FUNCTION_BLOCK Test_ListCountIncrements EXTENDS T_UnitTestBase
VAR
    List  : T_ListOfTests(Capacity := 10);
    Test0 : Test_ExampleTest;
END_VAR

METHOD RunTest
List.Clear();
List.AddTest(Test0);

AssertIsTrue(Condition := List.Count = 1,
             Message   := 'List.Count was not 1');

TestCompleted := TRUE;
END_METHOD

END_FUNCTION_BLOCK

(* stored: Version 1.1.0.1, ProductVersion 3.1.4024.12
   POU Test_ListCountIncrements: Id {4435a3b8-3ca9-4f28-8b70-83fec021bf80}, SpecialFunc None
   Method RunTest: Id {7d69c6e7-5ecd-40f0-afb8-6c5dace0a11b} *)
